(* PLC project PlcMain, Beckhoff Automation GmbH TwinCAT PLC Control 3.5.13.21 *)
(* stored: creationDateTime 2022-08-19T12:33:53.4229409, modificationDateTime 2022-08-19T12:33:53.4229409 *)

{attribute 'qualified_only'}
{attribute 'strict'}
TYPE State :
(
	Off,
	Busy,
	Ready,
	Done,
	Error,
	Setup
);
END_TYPE
